TYPE Result : INT; END_TYPE

(* stored: Version 1.1.0.1
   DUT Result: Id {0584450c-e377-4071-b6de-259ead2d47c1} *)
